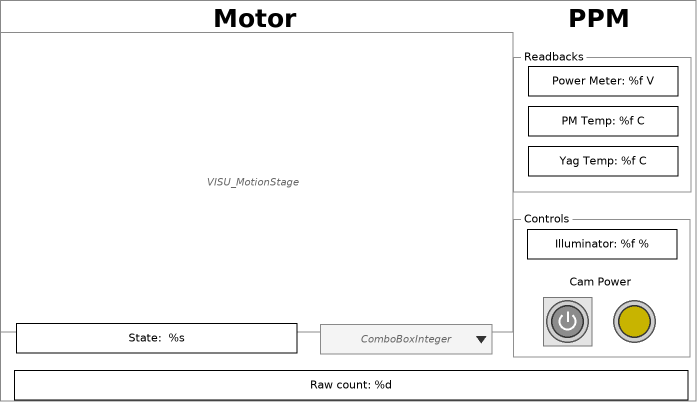
VISUALIZATION Visualization  // 697x402
    Label (14,3 482x30), "Motor"
    Label (503,3 192x30), "PPM"
    Rectangle (14,370 674x30), "Raw count: %d", text variable: Main.iAdjustedEncoder
    GroupBox (513,49 178x143), "Readbacks"
        Rectangle (15,17 150x30), "Power Meter: %f V", text variable: Main.fbPPM.fbPowerMeter.fVoltage
        Rectangle (15,57 150x30), "PM Temp: %f C", text variable: Main.fbPPM.fbPowerMeter.fbThermoCouple.fTemp
        Rectangle (15,97 150x30), "Yag Temp: %f C", text variable: Main.fbPPM.fbYagThermoCouple.fTemp
    GroupBox (513,211 177x146), "Controls"
        Rectangle (14,18 150x30), "Illuminator: %f %", text variable: Main.fbPPM.fbGige.fIlluminatorPercent
            OnMouseDown: write the text variable via Default, min 0, max 100
        Lamp1 (97,86 49x49), variable: Main.fbPPM.fbGige.bGigePower, style: Lamp-Lamp1-Yellow
        PowerSwitch (30,86 49x49), variable: Main.fbPPM.fbGige.bGigePower, behaviour: TOGGLE, style: Switch-PowerSwitch-Gray
        Label (9,56 157x30), "Cam Power"
    Frame (-7,32 520x300)
        shows VISU_MotionStage(VisuMotionStage := Main.M1, Extras := Main.M1_Extras)
    ComboBoxInteger (320,324 172x30), variable: Main.fbPPM.fbStates.enumSet, text list: 'TextListPPMStates'
    Rectangle (16,323 281x30), "State: %s", text variable: Main.fbPPM.fbStates.enumGet
END_VISUALIZATION

(* stored: Version 1.1.0.1, ProductVersion 3.1.4022.18
   Visu Visualization: Id {af2f16f4-e7e7-4019-a84a-cc323e4115d2} *)
